// Mitsubishi GX Works2 project: PLC 데이터 명령 (MOV)   PLC: Q03UDV

PROGRAM MAIN
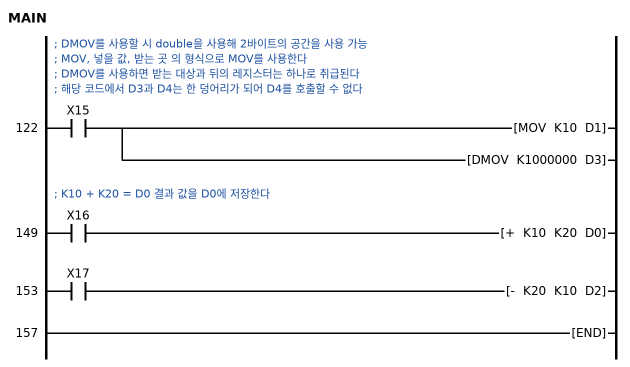
; DMOV를 사용할 시 double을 사용해 2바이트의 공간을 사용 가능
; MOV, 넣을 값, 받는 곳 의 형식으로 MOV를 사용한다
; DMOV를 사용하면 받는 대상과 뒤의 레지스터는 하나로 취급된다
; 해당 코드에서 D3과 D4는 한 덩어리가 되어 D4를 호출할 수 없다
122   LD      X15
      MOV     K10 D1
      DMOV    K1000000 D3
; K10 + K20 = D0 결과 값을 D0에 저장한다
149   LD      X16
      +       K10 K20 D0
153   LD      X17
      -       K20 K10 D2
157   END
END_PROGRAM
